{attribute 'qualified_only'}
{attribute 'strict'}
TYPE E_INSTANCE_CMD : // instructions for fb_Instance executions
(
	NULL,
  INIT,
  DISABLE,
  ENABLE,
  WORK,
  PROCEED := 100,
  FINISH,
  CLEAR
)UINT;
END_TYPE

(* stored: Version 1.1.0.1, ProductVersion 3.1.4024.15
   DUT E_INSTANCE_CMD: Id {fc824048-0a84-4d59-aced-c9bae584431d} *)
